RoboDK station: drilling.rdk

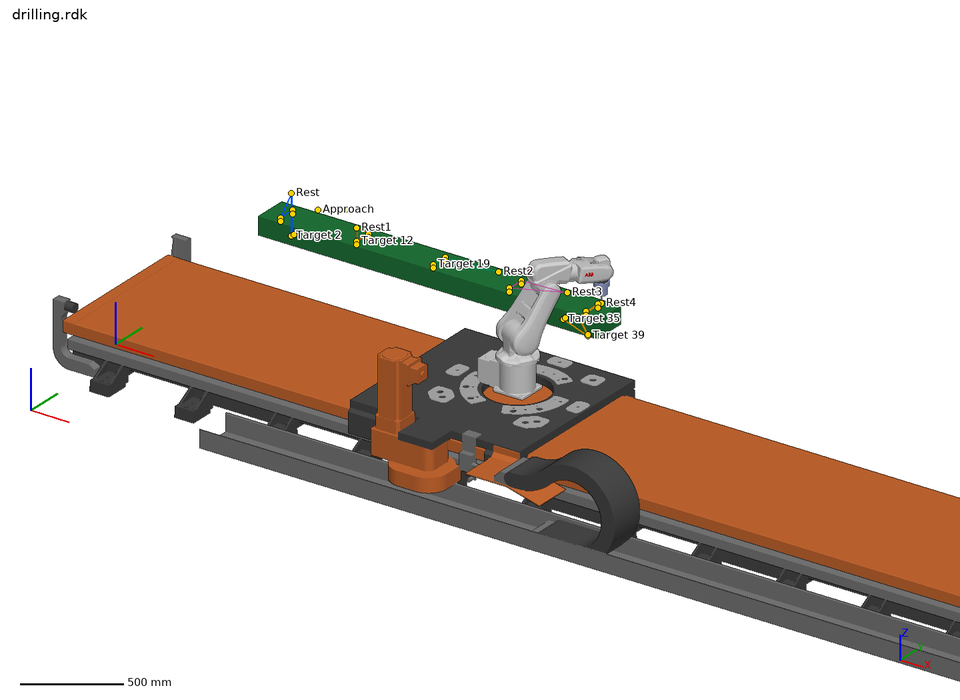
[picture v0: the station drawn from its stored meshes, robots at their saved joint values, targets as dots, program paths as lines]
Station template (saved by RoboDK 5.3.4). Poses are relative to the parent item; angles as X-Y-Z fixed-axis rotations.
  - frame ABB IRB 120-3/0.6 Base at (0, 0, 0) mm
  - frame worktable at (200, 480, 100) mm
    - object Task4_Part at (330, 1640, 460) mm, rotated rx 90 ry 0 rz 0 deg, size 2000 x 100 x 200 mm, geometry from Task4_Part.STL
    - target Approach (Cartesian target) at (933.5, 1086.8, 902.5) mm, rotated rx 0 ry 90 rz 0 deg; joints [0, 0, 0, 0, 0, 0] of ABB IRB 120-3/0.6
    - target Tape0 (joint target) at (445.5, 1086.8, 270.5) mm; joints [0] of ABB IRBT 4004 Standard 20m
    - target Target 2 (Cartesian target) at (530, 1440, 510) mm, rotated rx 0 ry 90 rz 90 deg; joints [63.189, 23.67, 64.627, -26.821, -88.48, 0.768] of ABB IRB 120-3/0.6
    - target Target 3 (Cartesian target) at (530, 1460, 510) mm, rotated rx 0 ry 90 rz 90 deg; joints [65.706, 25.284, 60.876, -24.342, -86.5, 1.582] of ABB IRB 120-3/0.6
    - target Target 5 (Cartesian target) at (430, 1490, 560) mm, rotated rx 180 ry 0 rz -93.01 deg; joints [92.227, 21.414, 3.902, 0, 64.684, 5.237] of ABB IRB 120-3/0.6
    - target Target 6 (Cartesian target) at (430, 1490, 540) mm, rotated rx 180 ry 0 rz -93.01 deg; joints [92.227, 22.45, 6.329, 0, 61.221, 5.237] of ABB IRB 120-3/0.6
    - target Target 7 (Cartesian target) at (430, 1590, 560) mm, rotated rx 180 ry 0 rz -93.01 deg; joints [91.783, 45.168, -31.22, 0, 76.052, 4.793] of ABB IRB 120-3/0.6
    - target Target 8 (Cartesian target) at (430, 1590, 540) mm, rotated rx 180 ry 0 rz -93.01 deg; joints [91.783, 45.436, -27.953, 0, 72.517, 4.793] of ABB IRB 120-3/0.6
    - target Rest (Cartesian target) at (530, 1440, 740) mm, rotated rx 0 ry 90 rz 90 deg; joints [63.189, -25.311, 50.763, -49.624, -36.305, 43.462] of ABB IRB 120-3/0.6
    - target Rest1 (Cartesian target) at (847.46, 1440, 740) mm, rotated rx 0 ry 90 rz 90 deg; joints [63.189, -25.311, 50.763, -49.624, -36.305, 43.462] of ABB IRB 120-3/0.6
    - target Tape1 (joint target) at (868.78, 1086.8, 270.5) mm; joints [223.28] of ABB IRBT 4004 Standard 20m
    - target Rest1 (Cartesian target) at (880, 1490, 630) mm, rotated rx 180 ry 0 rz -90 deg; joints [62.235, 32.387, -24.425, 0, 82.039, -27.765] of ABB IRB 120-3/0.6
    - target Target 12 (Cartesian target) at (880, 1490, 560) mm, rotated rx 180 ry 0 rz -90 deg; joints [62.235, 32.782, -12.038, 0, 69.257, -27.765] of ABB IRB 120-3/0.6
    - target Target 13 (Cartesian target) at (880, 1490, 540) mm, rotated rx -180 ry 0 rz -90 deg; joints [62.235, 33.538, -9.413, 0, 65.875, -27.765] of ABB IRB 120-3/0.6
    - target Target 14 (Cartesian target) at (880, 1590, 560) mm, rotated rx -180 ry 0 rz -90 deg; joints [67.148, 62.816, -61.331, 0, 88.515, -22.852] of ABB IRB 120-3/0.6
    - target Target 15 (Cartesian target) at (880, 1590, 540) mm, rotated rx 180 ry 0 rz -90 deg; joints [67.148, 60.821, -54.043, 0, 83.222, -22.852] of ABB IRB 120-3/0.6
    - target Tape2 (Cartesian target) at (1505.7, 1086.8, 270.5) mm; joints [1060.2] of ABB IRBT 4004 Standard 20m
    - target Rest2 (Cartesian target) at (1716.92, 1490, 630) mm, rotated rx 180 ry 0 rz -90 deg; joints [62.235, 32.387, -24.425, 0, 82.039, -27.765] of ABB IRB 120-3/0.6
    - target Target 19 (Cartesian target) at (1330, 1490, 560) mm, rotated rx 180 ry 0 rz -90 deg; joints [113.65, 29.277, -6.944, 0, 67.666, 23.65] of ABB IRB 120-3/0.6
    - target Target 20 (Cartesian target) at (1330, 1490, 540) mm, rotated rx 180 ry 0 rz -90 deg; joints [113.65, 30.131, -4.407, 0, 64.276, 23.65] of ABB IRB 120-3/0.6
    - target Target 21 (Cartesian target) at (1330, 1590, 560) mm, rotated rx 180 ry 0 rz -90 deg; joints [109.319, 55.633, -48.71, 0, 83.077, 19.319] of ABB IRB 120-3/0.6
    - target Target 22 (Cartesian target) at (1330, 1590, 540) mm, rotated rx 180 ry 0 rz -90 deg; joints [109.319, 55.043, -43.989, 0, 78.946, 19.319] of ABB IRB 120-3/0.6
    - target Tape3 (Cartesian target) at (1909.16, 1086.8, 270.5) mm; joints [1463.66] of ABB IRBT 4004 Standard 20m
    - target Rest3 (Cartesian target) at (2120.38, 1490, 630) mm, rotated rx 180 ry 0 rz -90 deg; joints [62.235, 32.387, -24.425, 0, 82.039, -27.765] of ABB IRB 120-3/0.6
    - target Target 25 (Cartesian target) at (1780, 1490, 560) mm, rotated rx 180 ry 0 rz -90 deg; joints [107.845, 25.661, -1.852, 0, 66.191, 17.845] of ABB IRB 120-3/0.6
    - target Target 26 (Cartesian target) at (1780, 1490, 540) mm, rotated rx 180 ry 0 rz -90 deg; joints [107.845, 26.604, 0.621, 0, 62.775, 17.845] of ABB IRB 120-3/0.6
    - target Target 27 (Cartesian target) at (1780, 1590, 560) mm, rotated rx 180 ry 0 rz -90 deg; joints [104.451, 50.337, -39.721, 0, 79.384, 14.451] of ABB IRB 120-3/0.6
    - target Target 28 (Cartesian target) at (1780, 1590, 540) mm, rotated rx 180 ry 0 rz -90 deg; joints [104.451, 50.271, -35.913, 0, 75.642, 14.451] of ABB IRB 120-3/0.6
    - target Tape4 (Cartesian target) at (2109.16, 1086.8, 270.5) mm; joints [1663.66] of ABB IRBT 4004 Standard 20m
    - target Rest4 (Cartesian target) at (2320.38, 1490, 630) mm, rotated rx 180 ry 0 rz -90 deg; joints [62.235, 32.352, -24.096, 0, 81.744, -27.765] of ABB IRB 120-3/0.6
    - target Target 31 (Cartesian target) at (2230, 1490, 560) mm, rotated rx 180 ry 0 rz -90 deg; joints [73.238, 25.191, -0.921, 0, 65.73, -16.762] of ABB IRB 120-3/0.6
    - target Target 32 (Cartesian target) at (2230, 1490, 540) mm, rotated rx 180 ry 0 rz -90 deg; joints [73.238, 26.165, 1.522, 0, 62.314, -16.762] of ABB IRB 120-3/0.6
    - target Target 33 (Cartesian target) at (2230, 1590, 560) mm, rotated rx 180 ry 0 rz -90 deg; joints [76.445, 49.624, -38.255, 0, 78.631, -13.555] of ABB IRB 120-3/0.6
    - target Target 34 (Cartesian target) at (2230, 1590, 540) mm, rotated rx 180 ry 0 rz -90 deg; joints [76.445, 49.642, -34.588, 0, 74.946, -13.555] of ABB IRB 120-3/0.6
    - target Target 35 (Cartesian target) at (2130, 1440, 510) mm, rotated rx 0 ry -90 rz -90 deg; joints [82.958, 20.758, 68.427, -7.043, -89.191, -179.9] of ABB IRB 120-3/0.6
    - target Target 36 (Cartesian target) at (2130, 1460, 510) mm, rotated rx 0 ry -90 rz -90 deg; joints [83.698, 22.585, 64.33, -6.311, -86.933, -179.661] of ABB IRB 120-3/0.6
    - target Target 37 (Cartesian target) at (2320.38, 1300, 630) mm, rotated rx 180 ry 0 rz -90 deg; joints [44.997, -2.315, 18.283, 0, 74.032, -45.003] of ABB IRB 120-3/0.6
    - target Target 39 (Cartesian target) at (2335.51, 1358.8, 510.08) mm, rotated rx 7.15 ry -89.99 rz -133.54 deg; joints [46.57, 20.75, 68.42, -7.04, -89.19, -179.9] of ABB IRB 120-3/0.6
    - target Target 41 (Cartesian target) at (2334.53, 1355, 517.81) mm, rotated rx -111.54 ry -82.78 rz -21.73 deg; joints [53.272, 14.439, 69.926, 6.441, -81.757, -173.915] of ABB IRB 120-3/0.6
  - frame ABB IRBT 4004 Standard 20m Base at (0, 1480, 0) mm
    - robot ABB IRBT 4004 Standard 20m: 1 axes, repeatability 0.1 mm
        modified DH rows (alpha deg, a mm, theta deg, d mm): 0, 0, 0, 0 linear
        base shift (645.5, 86.8, 370.5) mm, rotated rx 0 ry 90 rz 0 deg
        joint limits [0] to [20000]; home [0]; saved at [1663.66]
      - robot ABB IRB 120-3/0.6: 6 axes, payload 3 kg, reach 580 mm, repeatability 0.01 mm, weight 25 kg
          modified DH rows (alpha deg, a mm, theta deg, d mm): 0, 0, 0, 290; -90, 0, -90, 0; 0, 270, 0, 0; -90, 70, 0, 302; 90, 0, 0, 0; -90, 0, 180, 72
          joint limits [-165, -110, -90, -160, -120, -400] to [165, 110, 70, 160, 120, 400]; home [0, 0, 0, 0, 0, 0]; saved at [62.235, 32.352, -24.096, 0, 81.744, -27.765]
        - tool AssemblyDrillbit, TCP at (-2, 0, 112.5) mm, size 80 x 120 x 80 mm
  - program 程序10 (2 instructions, listed below)
  - program 程序1 (14 instructions, listed below)
  - program 程序2 (2 instructions, listed below)
  - program 程序3 (10 instructions, listed below)
  - program 程序4 (2 instructions, listed below)
  - program 程序5 (10 instructions, listed below)
  - program 程序6 (2 instructions, listed below)
  - program 程序7 (10 instructions, listed below)
  - program 程序8 (2 instructions, listed below)
  - program 程序9 (18 instructions, listed below)
  - program 主程序 (10 instructions, listed below)
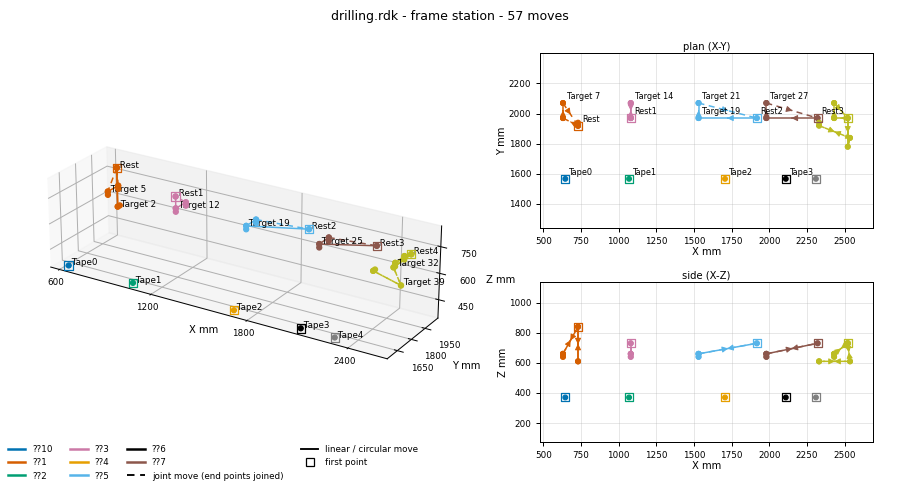
[picture p0: tool path of drilling.rdk in frame station, 57 of 57 moves have a stored position in this frame; points joined in program order, loops and branches not executed]

--- program 程序10 (robot ABB IRBT 4004 Standard 20m) ---
  设置参考: worktable
  MoveL (Tape0)

--- program 程序1 (robot ABB IRB 120-3/0.6) ---
  设置参考: worktable
  设置工具: AssemblyDrillbit
  MoveJ (Rest)
  MoveL (Target 2)
  MoveL (Target 3)
  MoveL (Target 2)
  MoveL (Rest)
  MoveJ (Target 5)
  MoveL (Target 6)
  MoveL (Target 5)
  MoveL (Target 7)
  MoveL (Target 8)
  MoveL (Target 7)
  MoveJ (Rest)

--- program 程序2 (robot ABB IRBT 4004 Standard 20m) ---
  设置参考: worktable
  MoveJ (Tape1)

--- program 程序3 (robot ABB IRB 120-3/0.6) ---
  设置参考: worktable
  设置工具: AssemblyDrillbit
  MoveJ (Rest1)
  MoveL (Target 12)
  MoveL (Target 13)
  MoveL (Target 12)
  MoveL (Target 14)
  MoveL (Target 15)
  MoveL (Target 14)
  MoveJ (Rest1)

--- program 程序4 (robot ABB IRBT 4004 Standard 20m) ---
  设置参考: worktable
  MoveL (Tape2)

--- program 程序5 (robot ABB IRB 120-3/0.6) ---
  设置参考: worktable
  设置工具: AssemblyDrillbit
  MoveJ (Rest2)
  MoveL (Target 19)
  MoveL (Target 20)
  MoveL (Target 19)
  MoveL (Target 21)
  MoveL (Target 22)
  MoveL (Target 21)
  MoveJ (Rest2)

--- program 程序6 (robot ABB IRBT 4004 Standard 20m) ---
  设置参考: worktable
  MoveJ (Tape3)

--- program 程序7 (robot ABB IRB 120-3/0.6) ---
  设置参考: worktable
  设置工具: AssemblyDrillbit
  MoveJ (Rest3)
  MoveL (Target 25)
  MoveL (Target 26)
  MoveL (Target 25)
  MoveL (Target 27)
  MoveL (Target 28)
  MoveL (Target 27)
  MoveJ (Rest3)

--- program 程序8 (robot ABB IRBT 4004 Standard 20m) ---
  设置参考: worktable
  MoveL (Tape4)

--- program 程序9 (robot ABB IRB 120-3/0.6) ---
  设置参考: worktable
  设置工具: AssemblyDrillbit
  MoveJ (Rest4)
  MoveL (Target 31)
  MoveL (Target 32)
  MoveL (Target 31)
  MoveL (Target 33)
  MoveL (Target 34)
  MoveL (Target 33)
  MoveJ (Rest4)
  MoveL (Target 37)
  MoveJ (Target 39)
  MoveJ (Target 35)
  MoveL (Target 36)
  MoveL (Target 35)
  MoveJ (Target 39)
  MoveJ (Target 37)
  MoveL (Rest4)

--- program 主程序 (robot ABB IRBT 4004 Standard 20m) ---
  调用 程序10
  调用 程序1
  调用 程序2
  调用 程序3
  调用 程序4
  调用 程序5
  调用 程序6
  调用 程序7
  调用 程序8
  调用 程序9
